// TIA Portal V17 export
// export: Created 2022-07-28T18:02:45.351851Z, ExportSetting None, DisplayName Totally Integrated Automation Portal, DisplayVersion V17, DisplayName TIA Portal Openness, DisplayVersion V17, DisplayName TIA Portal Teamcenter Gateway, DisplayVersion V17, DisplayName TIA Portal Version Control Interface, DisplayVersion V17, DisplayName TIA Portal Test Suite Advanced, DisplayVersion V17, DisplayName SINAMICS Startdrive Advanced, DisplayVersion V17, DisplayName SINAMICS DCC, DisplayVersion V17, DisplayName SINAMICS Startdrive G130, G150, S120, S150, SINAMICS MV, S210, DisplayVersion V17, DisplayName SINAMICS Startdrive G110M, G120, G120C, G120D, G120P, G115D, DisplayVersion V17, DisplayName STEP 7 Professional, DisplayVersion V17, DisplayName SIMATIC Energy Suite, DisplayVersion V17, DisplayName STEP 7 CFC, DisplayVersion V17, DisplayName STEP 7 Safety, DisplayVersion V17, DisplayName WinCC Advanced / Unified PC, DisplayVersion V17, DisplayName SIMATIC Visualization Architect, DisplayVersion V17
FUNCTION "Lib_FC_GenMoto_ChoiceCMD" : Void   // FC11, SCL
{ S7_Optimized_Access := 'TRUE' }
// stored: SetENOAutomatically false
   VAR_INPUT
      I_Mode : "UDT_Mode";   // Current mode
   END_VAR
   VAR_OUTPUT
      QI_CMD_Logic : Int;   // Command for use in logic
   END_VAR
   VAR_IN_OUT
      IQI_CMD_Global : Int;   // Command from global part
      IQI_CMD_Auto : Int;   // Command from auto part
      IQI_CMD_HMI : Int;   // Command from HMI for current element
   END_VAR
BEGIN
   //Reinit logic CMD
   #QI_CMD_Logic := 0;

   //Define CMD by priority modes
   IF #IQI_CMD_Global <> 0
   THEN
       #QI_CMD_Logic := #IQI_CMD_Global;
   ELSIF #I_Mode.Auto
   THEN
       IF #IQI_CMD_Auto <> 0
       THEN
           #QI_CMD_Logic := #IQI_CMD_Auto;
           #IQI_CMD_Auto := 0;
       ELSE
           #QI_CMD_Logic := #IQI_CMD_HMI;
           #IQI_CMD_HMI := 0;
       END_IF;
   ELSE
       IF #IQI_CMD_HMI <> 0
       THEN
           #QI_CMD_Logic := #IQI_CMD_HMI;
           #IQI_CMD_HMI := 0;
       ELSE
           #QI_CMD_Logic := #IQI_CMD_Auto;
           #IQI_CMD_Auto := 0;
       END_IF;
   END_IF;
END_FUNCTION
